TYPE ST_WinchStatus :
STRUCT
    fPositionMm : LREAL;
    xAxisEnabled : BOOL;
    eMode : E_WinchMode;
    xAlarmTravelLimit : BOOL;
    xAlarmEStop : BOOL;
    xAlarmEStopStopTimeout : BOOL;
    xAutoBusy : BOOL;
END_STRUCT
END_TYPE

(* stored: Version 1.1.0.1
   DUT ST_WinchStatus: Id {76f98901-64e9-46d5-8f8f-359cb26d7b2c} *)
